# EPICS substitutions: siteApps-725b29e158e8061764313f5708af9e46fe30c0a8/siteApps-725b29e158e8061764313f5708af9e46fe30c0a8/Tr1/tr1App/Db/userHost.substitutions
# Example substitutions file

file "db/dbExample1.db" {
    { user = "rootHost" }
}

file db/dbExample2.db {
    pattern { user, no, scan }
        { "rootHost", 1, "1 second" }
        { "rootHost", 2, "2 second" }
        { "rootHost", 3, "5 second" }
}
